# EPICS StreamDevice protocol: siteApps-725b29e158e8061764313f5708af9e46fe30c0a8/siteApps-725b29e158e8061764313f5708af9e46fe30c0a8/streamSim/protocols/streamsim.proto
# example stream protocol file

Terminator = CR LF;
ReplyTimeout = 10000; # 10 sec is very long, for keyboard input
ReadTimeout = 1000;   # also long for keyboard input

li {
    out "%(NAME)s?";
    in "%d";
}

lo {
    out "%(NAME)s=%i";
}
